// TIA Portal V21 export
VAR_GLOBAL   // PLC tag table "KAllSensore"
END_VAR
VAR_GLOBAL CONSTANT   // user constants
   KAllSens_Spare : Int := 1;   // Spare / Scorta
END_VAR
